// TIA Portal project "Motorsteuerung1.1 FC" (V17)

(* hardware
DEVICE "S7-300/ET200M-Station_1"  S7-300 station
   slot 0: "Profilschiene_0"  Rail  6ES7 390-1***0-0AA0
   slot 1: "PS 307 5A_1"  PS 307 5A  6ES7 307-1EA01-0AA0
   slot 2: "PLC_1"  CPU 314C-2 DP  6ES7 314-6CH04-0AB0  V3.3
      slot 0: "MPI-Schnittstelle_1"  MPI
      slot 1: "DP-Schnittstelle_1"  DP
      slot 2: "DI 24/DO 16_1"  DI24/DO16
      slot 3: "AI 5/AO 2_1"  AI5/AO2
      slot 4: "Zählen_1"  Counter
      slot 5: "Positionieren_1"  Positioning
   slot 4: "DI 16/DO 16x24VDC/0.5A_1"  DI16/DO16 x 24V / 0.5A  6ES7 323-1BL00-0AA0
   slot 5: "DI 16x24VDC_1"  DI16 x 24VDC  6ES7 321-1BH02-0AA0
   slot 6: "CP 342-5_1"  CP 342-5  6GK7 342-5DA03-0XE0  V6.0
   slot 7: "CP 343-1_1"  CP 343-1  6GK7 343-1EX30-0XE0  V2.0
*)

// ===== PLC "PLC_1"  CPU 314C-2 DP =====

VAR_GLOBAL   // PLC tag table "Motorsteuerung_Variablen"
   "M1_Start_Li" AT %E124.0 : Bool;   // Starttaster für Motor 1 im Linkslauf.
   "M1_Start_Re" AT %E124.1 : Bool;   // Starttaster für Motor 1 im Rechtslauf.
   "M1_Stop" AT %E124.2 : Bool;   // Stopptaster für Motor 1.
   "M1_Motorschutz_OK" AT %E124.3 : Bool;   // Motorschutz von Motor 1 ist betriebsbereit.
   "M2_Start_Li" AT %E125.0 : Bool;   // Starttaster für Motor 2 im Linkslauf.
   "M2_Start_Re" AT %E125.1 : Bool;   // Starttaster für Motor 2 im Rechtslauf.
   "M2_Stop" AT %E125.2 : Bool;   // Stopptaster für Motor 2.
   "M2_Motorschutz_OK" AT %E125.3 : Bool;   // Motorschutz von Motor 2 ist betriebsbereit.
   "Not_Aus" AT %E124.7 : Bool;   // Not-Aus für die gesamte Anlage.
   "M1_Ausgang_Li" AT %A124.0 : Bool;   // Ausgang für Motor 1 im Linkslauf.
   "M1_Ausgang_Re" AT %A124.1 : Bool;   // Ausgang für Motor 1 im Rechtslauf.
   "M2_Ausgang_Li" AT %A125.1 : Bool;   // Ausgang für Motor 2 im Linkslauf.
   "M2_Ausgang_Re" AT %A125.2 : Bool;   // Ausgang für Motor 2 im Rechtslauf.
END_VAR

DATA_BLOCK "Datenbaustein_1"   // DB1
{ S7_Optimized_Access := 'FALSE' }
VERSION : 0.1
   VAR
      Motor_1 : Struct
         Start_Li : Bool;
         Start_Re : Bool;
         Stop : Bool;
         Motorschutz : Bool;
         Ausgang_Li : Bool;
         Ausgang_Re : Bool;
         SR_Merker_Li : Bool;
         SR_Merker_Re : Bool;
      END_STRUCT;
      Motor_2 : Struct
         Start_Li : Bool;
         Start_Re : Bool;
         Stop : Bool;
         Motorschutz : Bool;
         Ausgang_Li : Bool;
         Ausgang_Re : Bool;
         SR_Merker_Li : Bool;
         SR_Merker_Re : Bool;
      END_STRUCT;
      Not_Aus : Bool;
   END_VAR
BEGIN
END_DATA_BLOCK

FUNCTION "Von" : Void   // FC1, FBD
TITLE = Absoluten Eingänge/Ausgänge Verbindung
{ S7_Optimized_Access := 'FALSE' }
VERSION : 0.1
// Ordnet die Signale der physischen Ein- und Ausgänge den Variablen des Datenbausteins zu.
BEGIN

REGION Network 1: Motor 1: Start_Li
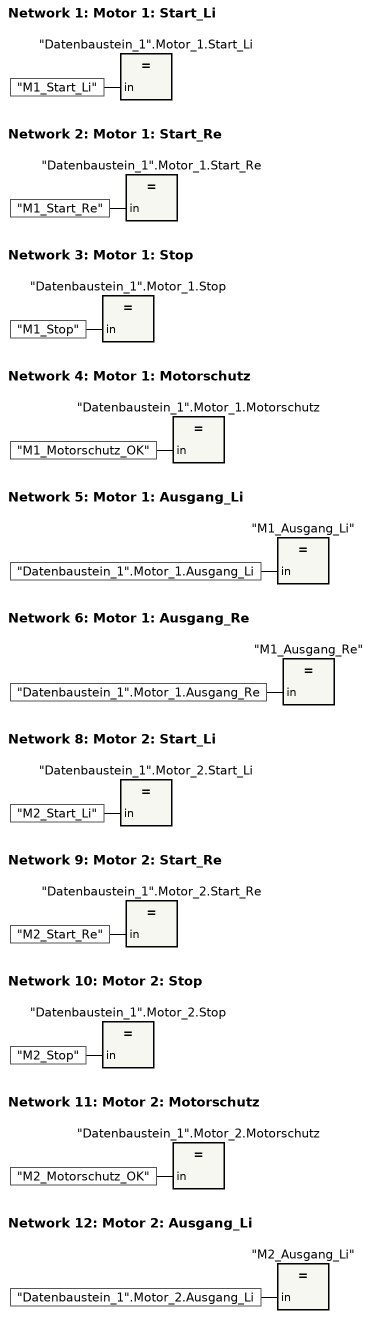
   "Datenbaustein_1".Motor_1.Start_Li := "M1_Start_Li";
END_REGION

REGION Network 2: Motor 1: Start_Re
   "Datenbaustein_1".Motor_1.Start_Re := "M1_Start_Re";
END_REGION

REGION Network 3: Motor 1: Stop
   "Datenbaustein_1".Motor_1.Stop := "M1_Stop";
END_REGION

REGION Network 4: Motor 1: Motorschutz
   "Datenbaustein_1".Motor_1.Motorschutz := "M1_Motorschutz_OK";
END_REGION

REGION Network 5: Motor 1: Ausgang_Li
   "M1_Ausgang_Li" := "Datenbaustein_1".Motor_1.Ausgang_Li;
END_REGION

REGION Network 6: Motor 1: Ausgang_Re
   "M1_Ausgang_Re" := "Datenbaustein_1".Motor_1.Ausgang_Re;
END_REGION

REGION Network 7: ///////////////////////////////////////////////////
END_REGION

REGION Network 8: Motor 2: Start_Li
   "Datenbaustein_1".Motor_2.Start_Li := "M2_Start_Li";
END_REGION

REGION Network 9: Motor 2: Start_Re
   "Datenbaustein_1".Motor_2.Start_Re := "M2_Start_Re";
END_REGION

REGION Network 10: Motor 2: Stop
   "Datenbaustein_1".Motor_2.Stop := "M2_Stop";
END_REGION

REGION Network 11: Motor 2: Motorschutz
   "Datenbaustein_1".Motor_2.Motorschutz := "M2_Motorschutz_OK";
END_REGION

REGION Network 12: Motor 2: Ausgang_Li
   "M2_Ausgang_Li" := "Datenbaustein_1".Motor_2.Ausgang_Li;
END_REGION

REGION Network 13: Motor 2: Ausgang_Re
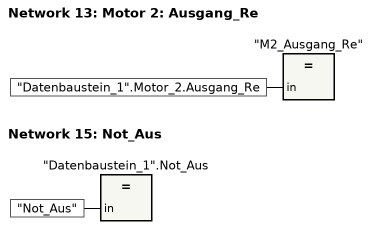
   "M2_Ausgang_Re" := "Datenbaustein_1".Motor_2.Ausgang_Re;
END_REGION

REGION Network 14: ///////////////////////////////////////////////////
END_REGION

REGION Network 15: Not_Aus
   "Datenbaustein_1".Not_Aus := "Not_Aus";
END_REGION
END_FUNCTION

FUNCTION "Motorsteuerung1.1" : Void   // FC50, FBD
TITLE = FC zur Steuerung eines Motors.
{ S7_Optimized_Access := 'FALSE' }
VERSION : 0.1
// Die Funktion übernimmt das Ein- und Ausschalten im Links- und Rechtslauf,
// überwacht Motorschutz und Not-Aus und verhindert einen direkten Richtungswechsel.
   VAR_INPUT
      Start_Li : Bool;
      Start_Re : Bool;
      Stop : Bool;
      Motorschutz_ok : Bool;
      Not_Aus : Bool;
   END_VAR
   VAR_OUTPUT
      Ausgang_Li : Bool;
      Ausgang_Re : Bool;
   END_VAR
   VAR_IN_OUT
      SR_Merker_Li : Bool;
      SR_Merker_Re : Bool;
   END_VAR
BEGIN

REGION Network 1: Linkslauf einschalten
   // Der Motor wird im Linkslauf gestartet.
   // Der Start ist nur möglich, wenn Stop, Not-Aus und Motorschutz freigegeben sind
   // und der Motor nicht bereits im Rechtslauf läuft.
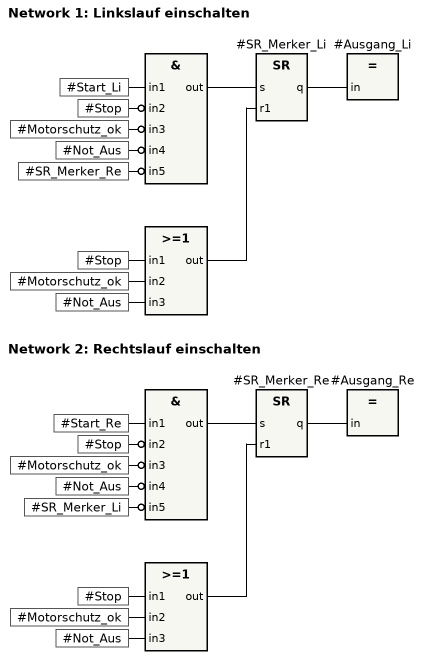
   IF #Start_Li AND NOT #Stop AND NOT #Motorschutz_ok AND NOT #Not_Aus AND NOT #SR_Merker_Re THEN
       #SR_Merker_Li := TRUE;   // SR flip-flop
   END_IF;
   IF #Stop OR #Motorschutz_ok OR #Not_Aus THEN #SR_Merker_Li := FALSE; END_IF;
   #Ausgang_Li := #SR_Merker_Li;
END_REGION

REGION Network 2: Rechtslauf einschalten
   // Der Motor wird im Rechtslauf gestartet.
   // Der Start ist nur möglich, wenn Stop, Not-Aus und Motorschutz freigegeben sind
   // und der Motor nicht bereits im Linkslauf läuft.
   IF #Start_Re AND NOT #Stop AND NOT #Motorschutz_ok AND NOT #Not_Aus AND NOT #SR_Merker_Li THEN
       #SR_Merker_Re := TRUE;   // SR flip-flop
   END_IF;
   IF #Stop OR #Motorschutz_ok OR #Not_Aus THEN #SR_Merker_Re := FALSE; END_IF;
   #Ausgang_Re := #SR_Merker_Re;
END_REGION
END_FUNCTION

ORGANIZATION_BLOCK "Main"   // OB1, FBD
TITLE = "Main Program Sweep (Cycle)" / Main Program Sweep (Cycle)
{ S7_Optimized_Access := 'FALSE' }
VERSION : 0.1
// Aufruf der Motorsteuerung für beide Motoren
// sowie Zuordnung der Ein- und Ausgänge.
   VAR_TEMP
      OB1_EV_CLASS : Byte;   // Bits 0-3 = 1 (Coming event), Bits 4-7 = 1 (Event class 1)
      OB1_SCAN_1 : Byte;   // 1 (Cold restart scan 1 of OB 1), 3 (Scan 2-n of OB 1)
      OB1_PRIORITY : Byte;   // Priority of OB Execution
      OB1_OB_NUMBR : Byte;   // 1 (Organization block 1, OB1)
      OB1_RESERVED_1 : Byte;   // Reserved for system
      OB1_RESERVED_2 : Byte;   // Reserved for system
      OB1_PREV_CYCLE : Int;   // Cycle time of previous OB1 scan (milliseconds)
      OB1_MIN_CYCLE : Int;   // Minimum cycle time of OB1 (milliseconds)
      OB1_MAX_CYCLE : Int;   // Maximum cycle time of OB1 (milliseconds)
      OB1_DATE_TIME : Date_And_Time;   // Date and time OB1 started
   END_VAR
BEGIN

REGION Network 1: Motor 1: Motorstartvorgang
   // Steuert den Motor 1 im Links- oder Rechtslauf.
   // Der Motor kann nur gestartet werden, wenn der Motorschutz freigegeben ist
   // und der Not-Aus nicht aktiv ist.
   // Ein Richtungswechsel ist nur nach Betätigung der Stop-Taste möglich.
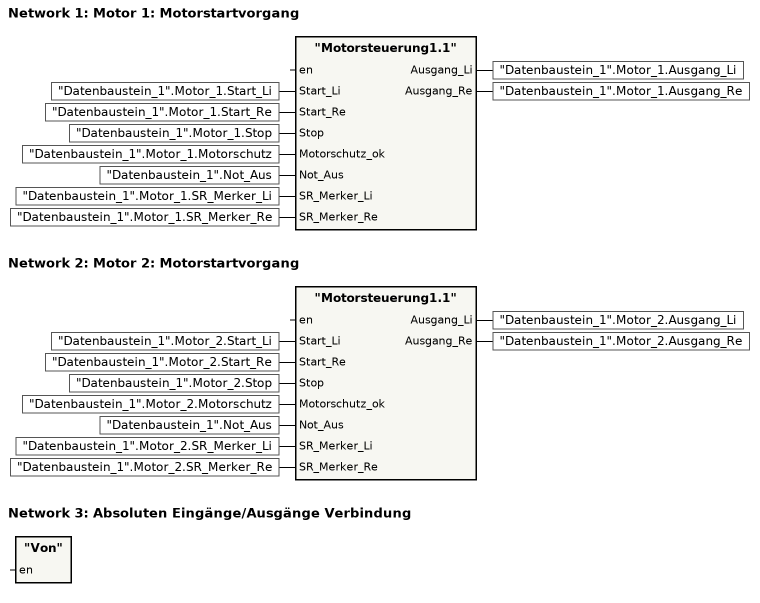
   "Motorsteuerung1.1"(Start_Li := "Datenbaustein_1".Motor_1.Start_Li,
                       Start_Re := "Datenbaustein_1".Motor_1.Start_Re,
                       Stop := "Datenbaustein_1".Motor_1.Stop,
                       Motorschutz_ok := "Datenbaustein_1".Motor_1.Motorschutz,
                       Not_Aus := "Datenbaustein_1".Not_Aus,
                       SR_Merker_Li := "Datenbaustein_1".Motor_1.SR_Merker_Li,
                       SR_Merker_Re := "Datenbaustein_1".Motor_1.SR_Merker_Re,
                       Ausgang_Li => "Datenbaustein_1".Motor_1.Ausgang_Li,
                       Ausgang_Re => "Datenbaustein_1".Motor_1.Ausgang_Re);
END_REGION

REGION Network 2: Motor 2: Motorstartvorgang
   // Steuert den Motor 2 im Links- oder Rechtslauf.
   // Der Motor kann nur gestartet werden, wenn der Motorschutz freigegeben ist
   // und der Not-Aus nicht aktiv ist.
   // Ein Richtungswechsel ist nur nach Betätigung der Stop-Taste möglich.
   "Motorsteuerung1.1"(Start_Li := "Datenbaustein_1".Motor_2.Start_Li,
                       Start_Re := "Datenbaustein_1".Motor_2.Start_Re,
                       Stop := "Datenbaustein_1".Motor_2.Stop,
                       Motorschutz_ok := "Datenbaustein_1".Motor_2.Motorschutz,
                       Not_Aus := "Datenbaustein_1".Not_Aus,
                       SR_Merker_Li := "Datenbaustein_1".Motor_2.SR_Merker_Li,
                       SR_Merker_Re := "Datenbaustein_1".Motor_2.SR_Merker_Re,
                       Ausgang_Li => "Datenbaustein_1".Motor_2.Ausgang_Li,
                       Ausgang_Re => "Datenbaustein_1".Motor_2.Ausgang_Re);
END_REGION

REGION Network 3: Absoluten Eingänge/Ausgänge Verbindung
   // Zuordnung der DB-Variablen zu den
   // physikalischen Ein- und Ausgängen.
   "Von"();
END_REGION
END_ORGANIZATION_BLOCK